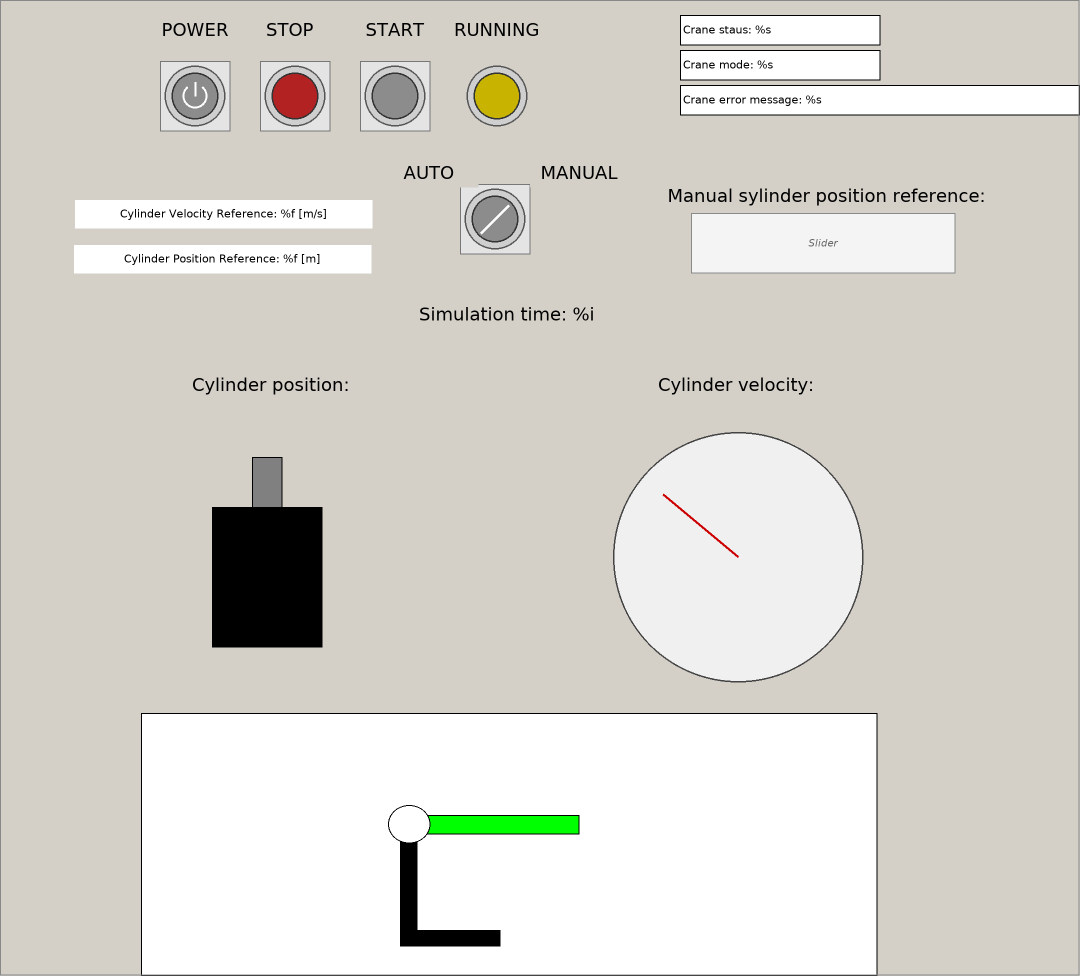
VISUALIZATION CraneHMI  // 1080x976
    PowerSwitch (160,61 70x70), variable: HMI.bPower, behaviour: TOGGLE, style: Switch-PowerSwitch-Gray
    RotarySwitch (460,184 70x70), variable: HMI.bMode, behaviour: TOGGLE, style: Switch-RotarySwitch-Gray
    PushSwitch (360,61 70x70), variable: HMI.bStart, behaviour: TOGGLE, style: Switch-PushSwitch-Gray
    Rectangle (145,16 100x28), "POWER"
    Rectangle (345,16 100x28), "START"
    Rectangle (380,159 98x28), "AUTO"
    Rectangle (530,159 98x28), "MANUAL"
    Lamp1 (462,61 70x70), variable: HMI.bRunning, style: Lamp-Lamp1-Yellow
    Rectangle (447,16 100x28), "RUNNING"
    Rectangle (239,301 536x27), "Simulation time: %i", text variable: CraneSimulation.fTime
    Meter360 (613,432 250x250), value: HMI.fCylinderVelocityReference, style: Meter-Meter360-Gray, scale format: %.2f, scale -0.05..0.05
    Rectangle (182,372 178x26), "Cylinder position:"
    Rectangle (647,372 178x26), "Cylinder velocity:"
    Rectangle (646,184 361x24), "Manual sylinder position reference:"
    Rectangle (680,85 400x30), "Crane error message: %s", text variable: HMI.sPistonEndStopMessage
    Rectangle (680,50 200x30), "Crane mode: %s", text variable: HMI.eCraneMode
    Rectangle (680,15 200x30), "Crane staus: %s", text variable: HMI.eCraneStatus
    Slider (691,213 264x60), variable: Inputs.fManualCylinderPositionReference, scale 0..0.5
    Rectangle (252,457 30x180)
        p2738717112: -HMI.fCylinderPositonReference*100
    Rectangle (212,507 110x140)
    Textfield (73,244 299x30), "Cylinder Position Reference: %f [m]", text variable: HMI.fCylinderPositonReference
    Textfield (74,199 299x30), "Cylinder Velocity Reference: %f [m/s]", text variable: HMI.fCylinderVelocityReference
        OnMouseClick: write the text variable via Default
    PushSwitch (260,61 70x70), variable: HMI.bStop, behaviour: TAP, style: Switch-PushSwitch-Red
    Rectangle (240,16 100x28), "STOP"
    Rectangle (141,713 736x263)
    Rectangle (400,930 100x16)
    Rectangle (400,810 17x130)
    Rectangle (409,815 170x19), angle 5
        p2858320360: -HMI.fBoomAngle
    Ellipse (388,805 42x38)
END_VISUALIZATION

(* stored: Version 1.1.0.1, ProductVersion 3.1.4024.10
   Visu CraneHMI: Id {b5520909-ac3e-4cb2-bbd3-14e4794d6a77} *)
